# EPICS substitutions: testApp/Db/cryocon.substitutions
global {p=\$(P)}

file "channel.template" {
{ P, CHANNEL }
{ "\$(P), "A" }
{ "\$(P), "B" }
{ "\$(P), "C" }
{ "\$(P), "D" }
{ "\$(P), "E" }
{ "\$(P), "F" }
{ "\$(P), "G" }
{ "\$(P), "H" }
}
